// TIA Portal V20 export
TYPE "LAxisCtrl_typePosAbsolute"
TITLE = LAxisCtrl_typePosAbsolute
// Support: tech.team.motioncontrol@siemens.com 
// Fax: +49 (0) 9131/98-1297
   STRUCT
      position : LReal := 0.0;   // Absolute target position
      velocity : LReal := -1.0;   // Velocity setpoint for absolute positioning (Value > 0.0: The specified value is used; Value = 0.0: Not permitted; Value < 0.0: Use of the default value configured in the technology object)
      acceleration : LReal := -1.0;   // Acceleration setpoint for absolute positioning (Value > 0.0: The specified value is used; Value = 0.0: Not permitted; Value < 0.0: Use of the default value configured in the technology object)
      deceleration : LReal := -1.0;   // Deceleration setpoint for absolute positioning (Value > 0.0: The specified value is used; Value = 0.0: Not permitted; Value < 0.0: Use of the default value configured in the technology object)
      jerk : LReal := -1.0;   // Jerk for absolute positioning (Value > 0.0: Smooth velocity profile, the specified value is used; (Value = 0.0: Trapezoid velocity profile; (Value < 0.0: Use of the default value configured in the technology object)
      direction : Int := 1;   // Motion direction of the axis (1: Positive direction; 2: Negative direction; 3: Shortest way)
      positionChangeOnTheFly : Bool := FALSE;   // TRUE: Changing position on-the-fly; FALSE: Position change requires a new rising edge at posAbsolute input
      velocityChangeOnTheFly : Bool := FALSE;   // TRUE: Changing velocity on-the-fly; FALSE: Velocity change requires a new rising edge at posAbsolute input
   END_STRUCT;
END_TYPE
